FUNCTION_BLOCK TEMPLATE_COMPFB
  (* Standard: 61499-2 *)
  (* Version 1.0, 11-01-12, GASR, Universidade do Estado de Santa Catarina *)
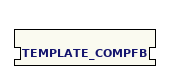
END_FUNCTION_BLOCK
